Staubli VAL3: stop.pgx

program stop()
begin
  clearBuffer(io:tcp_client)
  popUpMsg("Pending movement commands have been canceled")
  resetMotion()
end
